// TIA Portal V19 export
DATA_BLOCK "Gestion des sorties_DB"   // DB12
// stored: InstanceOfName Gestion des sorties, InstanceOfType FB
"Gestion des sorties"
BEGIN
END_DATA_BLOCK
